// /VISU_HELPER_Combobox_eControllerType
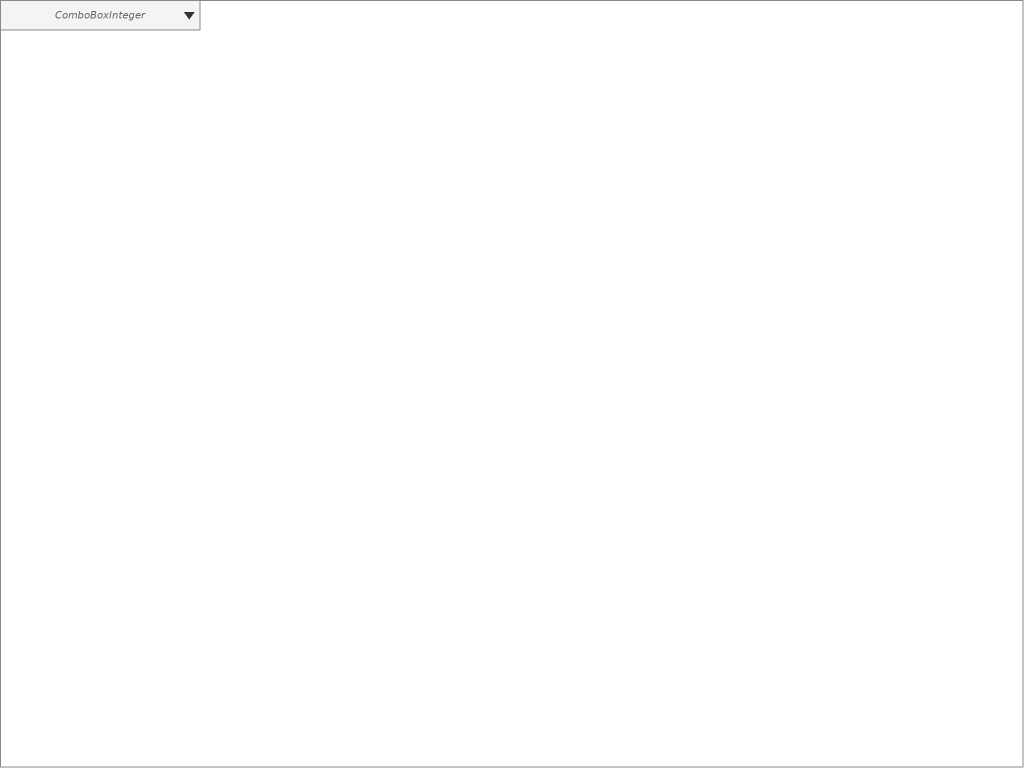
VISUALIZATION VISU_HELPER_Combobox_eControllerType  // 1024x768
VAR_IN_OUT
    varEnum : eControllerType;
END_VAR
    ComboBoxInteger (0,0 200x30), variable: varEnum, text list: 'TextListForCombobox_eControllerType'
END_VISUALIZATION

// /CS_VISU_PT2s
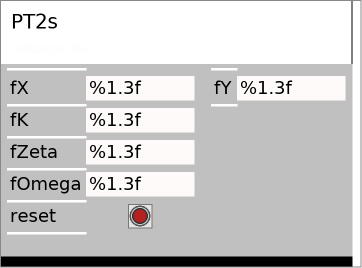
VISUALIZATION CS_VISU_PT2s  // 362x268
VAR_INPUT
   {attribute 'parameterstringof' := 'm_Input_FB'}
   m_Input_INST_Str : STRING;
END_VAR
VAR_IN_OUT
   m_Input_FB : PT2s;
END_VAR
    RoundedRectangle (0,0 352x81)
    RoundedRectangle (0,226 352x40)
    Rectangle (0,64 352x192)
    PushSwitch (128,204 24x24), variable: m_Input_FB.bReset, behaviour: TOGGLE, style: Switch-PushSwitch-Red
    Rectangle (8,8 352x27), "PT2s"
    Rectangle (8,35 352x27), "Instance: %s", text variable: m_Input_INST_Str
    Rectangle (7,68 79x2)
    Rectangle (86,76 108x24), "%1.3f", text variable: m_Input_FB.fX
        OnMouseClick: write the text variable via Default
    Rectangle (7,76 79x24), "fX"
    Rectangle (7,104 79x2)
    Rectangle (86,108 108x24), "%1.3f", text variable: m_Input_FB.fK
        OnMouseClick: write the text variable via Default
    Rectangle (7,108 79x24), "fK"
    Rectangle (7,136 79x2)
    Rectangle (86,140 108x24), "%1.3f", text variable: m_Input_FB.fZeta
        OnMouseClick: write the text variable via Default
    Rectangle (7,140 79x24), "fZeta"
    Rectangle (7,168 79x2)
    Rectangle (86,172 108x24), "%1.3f", text variable: m_Input_FB.fOmega
        OnMouseClick: write the text variable via Default
    Rectangle (7,172 79x24), "fOmega"
    Rectangle (7,200 79x2)
    Rectangle (7,204 79x24), "reset"
    Rectangle (7,232 79x2)
    Rectangle (211,68 26x2)
    Rectangle (237,76 108x24), "%1.3f", text variable: m_Input_FB.fY
    Rectangle (211,76 26x24), "fY"
    Rectangle (211,104 26x2)
END_VISUALIZATION

// /CS_VISU_Deadband
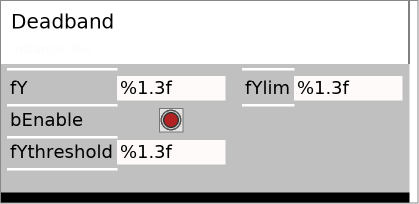
VISUALIZATION CS_VISU_Deadband  // 419x204
VAR_INPUT
   {attribute 'parameterstringof' := 'm_Input_FB'}
   m_Input_INST_Str : STRING;
END_VAR
VAR_IN_OUT
   m_Input_FB : Deadband;
END_VAR
    RoundedRectangle (0,0 409x81)
    RoundedRectangle (0,162 409x40)
    Rectangle (0,64 409x128)
    PushSwitch (159,108 24x24), variable: m_Input_FB.bEnable, behaviour: TOGGLE, style: Switch-PushSwitch-Red
    Rectangle (8,8 409x27), "Deadband"
    Rectangle (8,35 409x27), "Instance: %s", text variable: m_Input_INST_Str
    Rectangle (7,68 110x2)
    Rectangle (117,76 108x24), "%1.3f", text variable: m_Input_FB.fY
        OnMouseClick: write the text variable via Default
    Rectangle (7,76 110x24), "fY"
    Rectangle (7,104 110x2)
    Rectangle (7,108 110x24), "bEnable"
    Rectangle (7,136 110x2)
    Rectangle (117,140 108x24), "%1.3f", text variable: m_Input_FB.fYthreshold
        OnMouseClick: write the text variable via Default
    Rectangle (7,140 110x24), "fYthreshold"
    Rectangle (7,168 110x2)
    Rectangle (242,68 52x2)
    Rectangle (294,76 108x24), "%1.3f", text variable: m_Input_FB.fYlim
    Rectangle (242,76 52x24), "fYlim"
    Rectangle (242,104 52x2)
END_VISUALIZATION

(* text list TextListForCombobox_eSignalShape (id | default)
  1 | OFF
  2 | OFFSET
  3 | RECTANGLE
  4 | TRIANGLE
  5 | SINUS
  6 | RAMP
   |  *)

(* text list TextListForCombobox_eControllerType (id | default)
  1 | P
  2 | I
  3 | PI
  4 | PDT1
  5 | PIDT1
   |  *)
